INTERFACE I_String_Builder EXTENDS T_Query_Interface

// Number of bytes allocated in memory for the string builder's contents.
PROPERTY _Capacity : T_Size
GET
END_GET
END_PROPERTY

// Current size of string builder contents
PROPERTY _Length : T_Size
GET
END_GET
END_PROPERTY

// Appends the given string to the end of the string builder's contents.
METHOD Append : I_String_Builder
VAR_INPUT
	sValue : T_Long_String;
END_VAR
END_METHOD

// Appends the given value to the end of the string builder's contents.
METHOD Append_Any : I_String_Builder
VAR_INPUT
	Value : ANY;
END_VAR
END_METHOD

// !!!UNSAFE!!! THIS WILL APPEND UP TO THE NULL CHARACTER. IF NO NULL EXISTS, THIS WILL RUN FOREVER!
// | Append raw values directly to the internal string buffer. This is meant for appending dynamic strings to the string builder.
METHOD Append_Buffer : I_String_Builder
VAR_INPUT
	pBuffer : POINTER TO BYTE;
END_VAR
END_METHOD

// Appends a new line (\r\n or $r$n) to string builder's contents.
METHOD Append_Line : I_String_Builder
END_METHOD

// Empties the string builder's contents, resetting its length to zero.
METHOD Clear : I_String_Builder
END_METHOD

// Copies a subset of characters in the string builder from specified position at specified length to a string
METHOD Copy_Substring_To : I_String_Builder
VAR_INPUT
	Position, Length : T_Size;
	Value : ANY;
END_VAR
END_METHOD

// Copies contents of string builder to given string of any size
METHOD Copy_To : I_String_Builder
VAR_INPUT
	Value : ANY;
END_VAR
END_METHOD

// !!!UNSAFE!!! DON'T FORGET TO RELEASE/DELETE FROM	MEMORY WHEN DONE!
// | Get a copy of the internal string buffer at the size of the string length + 1.
METHOD Get_Buffer : I_String_Builder
VAR_IN_OUT
	pBuffer : POINTER TO BYTE;
END_VAR
END_METHOD

// Retrieves the number of bytes allocated in memory for the string builder's contents.
METHOD Get_Capacity : I_String_Builder
VAR_OUTPUT
	Capacity : T_Size;
END_VAR
END_METHOD

// Gets character at specified position in the string builder
METHOD Get_Char : T_Char
VAR_INPUT
	Position : T_Size;
END_VAR
END_METHOD

// Retrieves the current size of string builder contents
METHOD Get_Length : I_String_Builder
VAR_OUTPUT
	Length : T_Size;
END_VAR
END_METHOD

// Converts contents of string builder to string and returns them
METHOD Get_String : T_Long_String
VAR_INPUT
END_VAR
END_METHOD

// Get a subset of characters in the string builder from specified position at specified length and returns them as a string
METHOD Get_Substring : T_Long_String
VAR_INPUT
	Position, Length : T_Size;
END_VAR
END_METHOD

// Inserts the given string at the specified position.
METHOD Insert : I_String_Builder
VAR_INPUT
	Position : T_Size;
	sValue : T_Long_String;
END_VAR
END_METHOD

// Inserts the given value at the specified position.
METHOD Insert_Any : I_String_Builder
VAR_INPUT
	Position : T_Size;
	Value : ANY;
END_VAR
END_METHOD

// !!!UNSAFE!!! THIS WILL INSERT UP TO THE NULL CHARACTER. IF NO NULL EXISTS, THIS WILL RUN FOREVER!
// | Inserts raw values directly to the internal string buffer at the specified position. This is meant for inserting dynamic strings to the string builder.
METHOD Insert_Buffer : I_String_Builder
VAR_INPUT
	Position : T_Size;
	pBuffer : POINTER TO BYTE;
END_VAR
END_METHOD

// Joins/Merges the string contents of the current string builder with that on the specified string builder at the specified position
METHOD Join : I_String_Builder
VAR_INPUT
	Position : T_Size;
	ipString_Builder : I_String_Builder;
END_VAR
END_METHOD

// Removes the characters in the string builder from specified position at specified length.
METHOD Remove : I_String_Builder
VAR_INPUT
	Position, Length : T_Size;
END_VAR
END_METHOD

// Replaces the instance of the old string in the string builder with the new string.
// If bReplace_All = TRUE, all instances of the old string are placed, else only the first instance.
METHOD Replace : I_String_Builder
VAR_INPUT
	sOld_Value,
	sNew_Value : T_Long_String;
	bReplace_All : BOOL;
END_VAR
END_METHOD

// Replaces the instance of the old value in the string builder with the new value.
// If bReplace_All = TRUE, all instances of the old value are placed, else only the first instance.
METHOD Replace_Any : I_String_Builder
VAR_INPUT
	Old_Value : ANY;
	New_Value : ANY;
	bReplace_All : BOOL;
END_VAR
END_METHOD

// Reverses the string contents in the string builder
METHOD Reverse : I_String_Builder
VAR_INPUT
END_VAR
END_METHOD

// Finds the position of the first instance of a given string in the content's of the string builder from a starting position
METHOD Search : I_String_Builder
VAR_INPUT
	sValue : T_Long_String;
	Start_Position : T_Size;
END_VAR
VAR_OUTPUT
	Position : T_Size;
END_VAR
END_METHOD

// Finds the position of the first instance of a given value in the content's of the string builder from a starting position
METHOD Search_Any : I_String_Builder
VAR_INPUT
	Value : ANY;
	Start_Position : T_Size;
END_VAR
VAR_OUTPUT
	Position : T_Size := -1;
END_VAR
END_METHOD

// Appends selected characters from the current string builder to the selected string builder
METHOD Split : I_String_Builder
VAR_INPUT
	Position, Length : T_Size;
	ipString_Builder : I_String_Builder;
END_VAR
END_METHOD

// Reduces the capacity of the string builder to match the size of its contents, potentially reducing memory usage.
METHOD Strink_To_Fit : I_String_Builder
END_METHOD

// Converts all alphabetic characters in string builder to lowercase characters
METHOD To_Lower_Case : I_String_Builder
VAR_INPUT
END_VAR
END_METHOD

// Converts all alphabetic characters in string builder to uppercase characters
METHOD To_Upper_Case : I_String_Builder
VAR_INPUT
END_VAR
END_METHOD

// Removes all ASCII white space (spaces, tabs, carriage returns, and linefeeds) from the beginning, end, or both ends of string in the string builder
METHOD Trim_Whitespace : I_String_Builder
VAR_INPUT
	Location : T_Whitespace_Location;
END_VAR
END_METHOD

END_INTERFACE

(* stored: Version 1.1.0.1, ProductVersion 3.1.4024.4
   Itf I_String_Builder: Id {0720aa24-e3c8-41ae-a5a5-43696928f33d}
   Property _Capacity: Id {ba2a03c7-3755-45be-9ba0-4cd7e9d4b654}
   Get Get: Id {8b2c5724-7fcd-4312-ad6e-a12bb686f67a}
   Property _Length: Id {17c1e06b-941b-4841-91af-8cf372a9402d}
   Get Get: Id {30c9a3b2-a463-49ec-9f49-8a6f9e9842d0}
   Method Append: Id {19b8fae6-09f3-4d84-ae29-bb5020725b33}
   Method Append_Any: Id {48ff2b13-1615-43d0-8ea1-f6da83400a8a}
   Method Append_Buffer: Id {701bace9-44d5-460e-854d-cf9549386309}
   Method Append_Line: Id {553d213b-d668-4f2a-9e90-9a4310ae582e}
   Method Clear: Id {32a55980-f511-4d0d-a0d0-7301b9fbdbb4}
   Method Copy_Substring_To: Id {4c3595ba-6ba9-4731-ae1c-879194d0db68}
   Method Copy_To: Id {49378fb5-1ade-4d07-8b6c-a6431d528a2f}
   Method Get_Buffer: Id {63f9469e-26fb-436a-960f-f6adebffafe5}
   Method Get_Capacity: Id {71cbf03d-e226-420a-834e-72ffc3932270}
   Method Get_Char: Id {3e52b663-ff3f-47bb-b31c-eb04589f1b2c}
   Method Get_Length: Id {4d75dca5-6846-48de-9ae9-a24748a2ac1e}
   Method Get_String: Id {8301de19-c685-4e69-9b85-2430eb94ce14}
   Method Get_Substring: Id {8a394a0a-1e9a-42e5-9e2d-10f694d3cc8b}
   Method Insert: Id {05c3b0b6-cd11-49d2-991c-d9cf83dd2683}
   Method Insert_Any: Id {a5d890d0-ef2b-486c-9e2b-33a80ca46291}
   Method Insert_Buffer: Id {bace6fdb-8718-48f8-aa66-cd4b176d295e}
   Method Join: Id {d0a233f9-ffd4-4203-a624-e6d118b02fac}
   Method Remove: Id {812add6f-98c2-4955-8bd6-1a170155baf7}
   Method Replace: Id {e7e1e1b7-6e39-4983-8c57-829e9b04283e}
   Method Replace_Any: Id {4aca1964-ebf7-4a81-bf85-1203ad4e0c3d}
   Method Reverse: Id {d87f1fbf-11bb-4f80-9977-10b6848e2685}
   Method Search: Id {745197dc-b26d-4ce6-a64b-6e5f96d9b7bd}
   Method Search_Any: Id {123176dc-8ab6-4b6d-8fc6-479209e1aa55}
   Method Split: Id {d9a27e86-600a-4dac-a484-7322fdc46d5c}
   Method Strink_To_Fit: Id {071ba2b7-38d2-4267-be28-53ec29f36e1f}
   Method To_Lower_Case: Id {6513716f-70f4-45e0-991c-ec8d32177933}
   Method To_Upper_Case: Id {18bacf23-80be-4f43-a001-26ceb23edef2}
   Method Trim_Whitespace: Id {e240cb29-e5ac-4610-9df5-6fc2bee97f04} *)
